PROGRAM BO02PL_LineBackground
VAR
END_VAR

MAIN.stLine_BO02PL.fbLine(stLine:=MAIN.stLine_BO02PL);
MAIN.stLine_BO02PL.stStation_BO02PL01.fbStation(
				stLine:=MAIN.stLine_BO02PL,
				stStation:=MAIN.stLine_BO02PL.stStation_BO02PL01);
MAIN.stLine_BO02PL.stStation_BO02PL02.fbStation(
				stLine:=MAIN.stLine_BO02PL,
				stStation:=MAIN.stLine_BO02PL.stStation_BO02PL02);

END_PROGRAM

(* stored: Version 1.1.0.1, ProductVersion 3.1.4024.15
   POU BO02PL_LineBackground: Id {9fb14285-6030-4043-bb7f-894388949805}, SpecialFunc None *)
